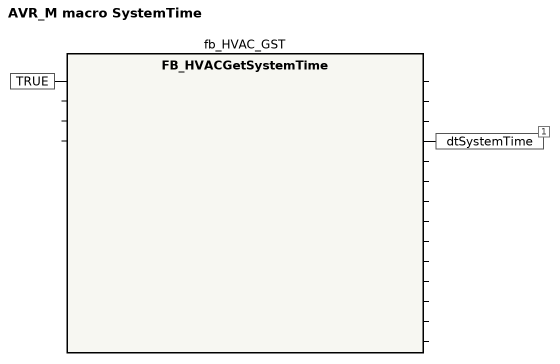
_CFC_ (* Continuous Function Chart, elements in execution order *)
#0 AND(SCHU_P2_2_UST_RE_PUSK, NOT SCHU_P2_2_YA1_DI6_ZKR)
#1 RT_T:R_TRIG(CLK: TRUE)
#2 OR(#1.Q, SCHU_P2_2_AVR_KOM_A)
#3 OR(SCHU_P2_2_AVR_KOM_M, NOT SCHU_P2_2_SA8_DI3_A, NOT SCHU_P2_2_SA1_DI5_A)
#4 TON_VKL:TON(IN: #3, PT: T#100ms)
#5 RS_avr_kom:RS(SET: #2, RESET1: #4.Q)
#6 TON_PUSK:TON(IN: #0, PT: t#6S)
#7 RT_Pusk:R_TRIG(CLK: #6.Q)
#8 OR(SCHU_P2_2_UST_RE_STOP, SCHU_P2_2_UST_RE_OSTANOV)
#9 RS_Pusk:RS(SET: #7.Q, RESET1: #8)
#10 SEL(#9.Q1, 0, 1)
#11 fb_HVACRC:FB_HVACRedundancyCtrl(EN: #5.Q1, eHVACDataSecurityType_Idle, FALSE, #10, NOT M1_OTKAZ, NOT M2_OTKAZ, -, -, -, -, -, -, SCHU_P2_2_MP2_2_1_DI3_RUN, SCHU_P2_2_MP2_2_2_DI7_RUN, -, -, -, -, -, -, -, dtSystemTime, -, SCHU_P2_2_M_SB_NAR, SCHU_P2_2_M_SB_NAR, SCHU_P2_2_SB, rHours, uiCount, overlap1Actuator, maxOnLevel, delayFBC)
#12 S SCHU_P2_2_AVR_A <= #11.ENO
#13 error <= #11.out 10
#14 NOT(#11.ENO)
#15 R SCHU_P2_2_AVR_A <= #14
#16 SCHU_P2_2_AVR_M <= #14
#17 AND(#11.ENO, #11.out 1)
#18 M1_PUSK <= #17
#19 AND(#11.ENO, #11.out 2)
#20 M2_PUSK <= #19
#21 MACRO SystemTime()
	#22 fb_HVAC_GST:FB_HVACGetSystemTime(TRUE, -, -, -)
	#23 dtSystemTime <= #22.out 4
END_MACRO
_END_CFC_
END_PROGRAM

(* POU TZBiS/TZB/Z_GVS1_Otk, CFC *)
PROGRAM Z_GVS1_Otk
VAR
	TON_YA2_OTKAZ: TON;
	SR_GVS1_Otkaz: SR;
	TON_YA2_Z_ZAM: TON;
END_VAR
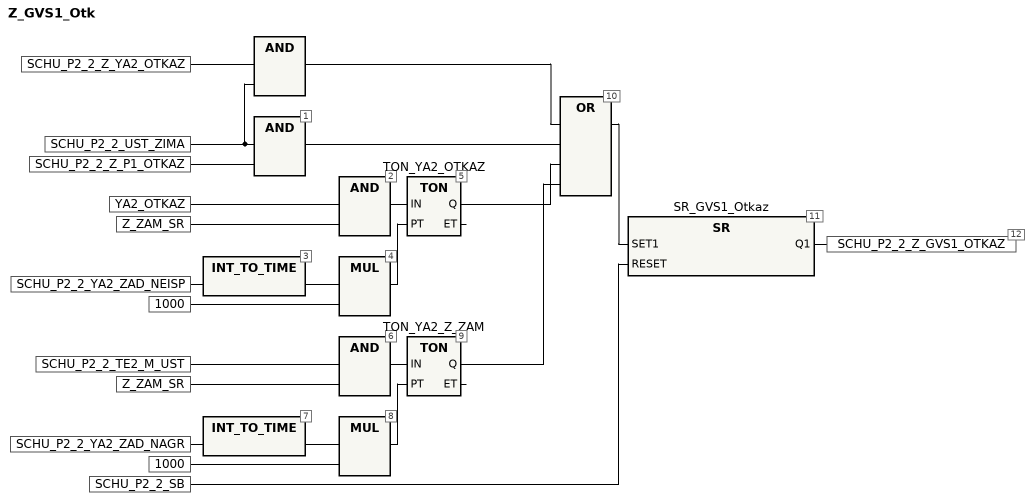
_CFC_ (* Continuous Function Chart, elements in execution order *)
#0 AND(SCHU_P2_2_Z_YA2_OTKAZ, SCHU_P2_2_UST_ZIMA)
#1 AND(SCHU_P2_2_UST_ZIMA, SCHU_P2_2_Z_P1_OTKAZ)
#2 AND(YA2_OTKAZ, Z_ZAM_SR)
#3 INT_TO_TIME(SCHU_P2_2_YA2_ZAD_NEISP)
#4 MUL(#3, 1000)
#5 TON_YA2_OTKAZ:TON(IN: #2, PT: #4)
#6 AND(SCHU_P2_2_TE2_M_UST, Z_ZAM_SR)
#7 INT_TO_TIME(SCHU_P2_2_YA2_ZAD_NAGR)
#8 MUL(#7, 1000)
#9 TON_YA2_Z_ZAM:TON(IN: #6, PT: #8)
#10 OR(#0, #1, #5.Q, #9.Q)
#11 SR_GVS1_Otkaz:SR(SET1: #10, RESET: SCHU_P2_2_SB)
#12 SCHU_P2_2_Z_GVS1_OTKAZ <= #11.Q1
_END_CFC_
(* the same logic as Structured Text *)
TON_YA2_OTKAZ(IN := YA2_OTKAZ AND Z_ZAM_SR, PT := INT_TO_TIME(SCHU_P2_2_YA2_ZAD_NEISP) * 1000);
TON_YA2_Z_ZAM(IN := SCHU_P2_2_TE2_M_UST AND Z_ZAM_SR, PT := INT_TO_TIME(SCHU_P2_2_YA2_ZAD_NAGR) * 1000);
SR_GVS1_Otkaz(SET1 := (SCHU_P2_2_Z_YA2_OTKAZ AND SCHU_P2_2_UST_ZIMA) OR (SCHU_P2_2_UST_ZIMA AND SCHU_P2_2_Z_P1_OTKAZ) OR TON_YA2_OTKAZ.Q OR TON_YA2_Z_ZAM.Q, RESET := SCHU_P2_2_SB);
SCHU_P2_2_Z_GVS1_OTKAZ := SR_GVS1_Otkaz.Q1;
END_PROGRAM

(* POU TZBiS/TZB/Z_M1_Avar, CFC *)
PROGRAM Z_M1_Avar
VAR
	SR_M1_Avar: SR;
END_VAR
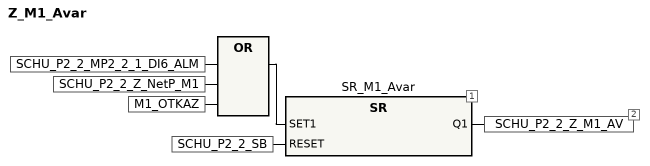
_CFC_ (* Continuous Function Chart, elements in execution order *)
#0 OR(SCHU_P2_2_MP2_2_1_DI6_ALM, SCHU_P2_2_Z_NetP_M1, M1_OTKAZ)
#1 SR_M1_Avar:SR(SET1: #0, RESET: SCHU_P2_2_SB)
#2 SCHU_P2_2_Z_M1_AV <= #1.Q1
_END_CFC_
(* the same logic as Structured Text *)
SR_M1_Avar(SET1 := SCHU_P2_2_MP2_2_1_DI6_ALM OR SCHU_P2_2_Z_NetP_M1 OR M1_OTKAZ, RESET := SCHU_P2_2_SB);
SCHU_P2_2_Z_M1_AV := SR_M1_Avar.Q1;
END_PROGRAM

(* POU TZBiS/TZB/Z_M1_NP, CFC *)
PROGRAM Z_M1_NP
VAR
	SR_M1_NPit: SR;
END_VAR
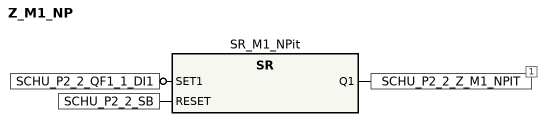
_CFC_ (* Continuous Function Chart, elements in execution order *)
#0 SR_M1_NPit:SR(SET1: NOT SCHU_P2_2_QF1_1_DI1, RESET: SCHU_P2_2_SB)
#1 SCHU_P2_2_Z_M1_NPIT <= #0.Q1
_END_CFC_
(* the same logic as Structured Text *)
SR_M1_NPit(SET1 := NOT SCHU_P2_2_QF1_1_DI1, RESET := SCHU_P2_2_SB);
SCHU_P2_2_Z_M1_NPIT := SR_M1_NPit.Q1;
END_PROGRAM

(* POU TZBiS/TZB/Z_M1_Pereg, CFC *)
PROGRAM Z_M1_Pereg
VAR
	SR_SCHU_P2_2_TSMP2_2_1_DI7: SR;
	TOF_TSMP1: TOF;
	TON1: TON;
END_VAR
VAR (* helpers for the ST form of the networks *)
	_t23 : BOOL;
END_VAR
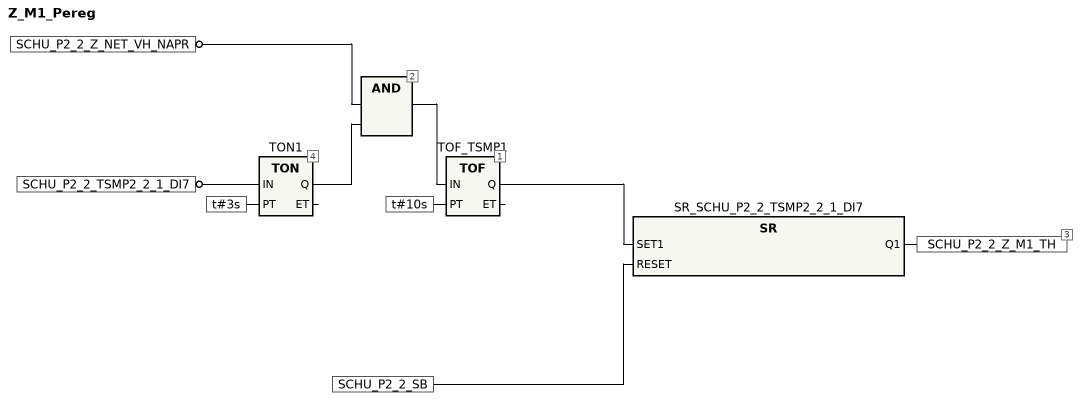
_CFC_ (* Continuous Function Chart, elements in execution order *)
#0 SR_SCHU_P2_2_TSMP2_2_1_DI7:SR(SET1: #1.Q, RESET: SCHU_P2_2_SB)
#1 TOF_TSMP1:TOF(IN: #2, PT: t#10s)
#2 AND(NOT SCHU_P2_2_Z_NET_VH_NAPR, #4.Q)
#3 SCHU_P2_2_Z_M1_TH <= #0.Q1
#4 TON1:TON(IN: NOT SCHU_P2_2_TSMP2_2_1_DI7, PT: t#3s)
_END_CFC_
(* the same logic as Structured Text *)
SR_SCHU_P2_2_TSMP2_2_1_DI7(SET1 := TOF_TSMP1.Q, RESET := SCHU_P2_2_SB);
TOF_TSMP1(IN := _t23, PT := t#10s);
_t23 := NOT SCHU_P2_2_Z_NET_VH_NAPR AND TON1.Q;
SCHU_P2_2_Z_M1_TH := SR_SCHU_P2_2_TSMP2_2_1_DI7.Q1;
TON1(IN := NOT SCHU_P2_2_TSMP2_2_1_DI7, PT := t#3s);
END_PROGRAM

(* POU TZBiS/TZB/Z_M2_Avar, CFC *)
PROGRAM Z_M2_Avar
VAR
	SR_M2_Avar: SR;
END_VAR
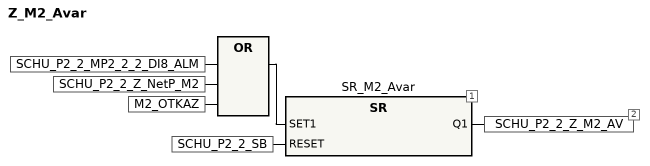
_CFC_ (* Continuous Function Chart, elements in execution order *)
#0 OR(SCHU_P2_2_MP2_2_2_DI8_ALM, SCHU_P2_2_Z_NetP_M2, M2_OTKAZ)
#1 SR_M2_Avar:SR(SET1: #0, RESET: SCHU_P2_2_SB)
#2 SCHU_P2_2_Z_M2_AV <= #1.Q1
_END_CFC_
(* the same logic as Structured Text *)
SR_M2_Avar(SET1 := SCHU_P2_2_MP2_2_2_DI8_ALM OR SCHU_P2_2_Z_NetP_M2 OR M2_OTKAZ, RESET := SCHU_P2_2_SB);
SCHU_P2_2_Z_M2_AV := SR_M2_Avar.Q1;
END_PROGRAM

(* POU TZBiS/TZB/Z_M2_NP, CFC *)
PROGRAM Z_M2_NP
VAR
	SR_M2_NPit: SR;
END_VAR
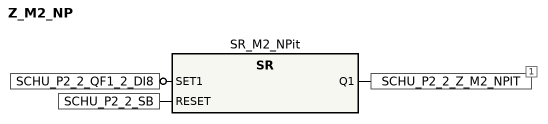
_CFC_ (* Continuous Function Chart, elements in execution order *)
#0 SR_M2_NPit:SR(SET1: NOT SCHU_P2_2_QF1_2_DI8, RESET: SCHU_P2_2_SB)
#1 SCHU_P2_2_Z_M2_NPIT <= #0.Q1
_END_CFC_
(* the same logic as Structured Text *)
SR_M2_NPit(SET1 := NOT SCHU_P2_2_QF1_2_DI8, RESET := SCHU_P2_2_SB);
SCHU_P2_2_Z_M2_NPIT := SR_M2_NPit.Q1;
END_PROGRAM

(* POU TZBiS/TZB/Z_M2_Pereg, CFC *)
PROGRAM Z_M2_Pereg
VAR
	SR_SCHU_P2_2_TSMP2_2_2_DI1: SR;

	TOF_TSMP2: TOF;
	TON1: TON;
END_VAR
VAR (* helpers for the ST form of the networks *)
	_t28 : BOOL;
END_VAR
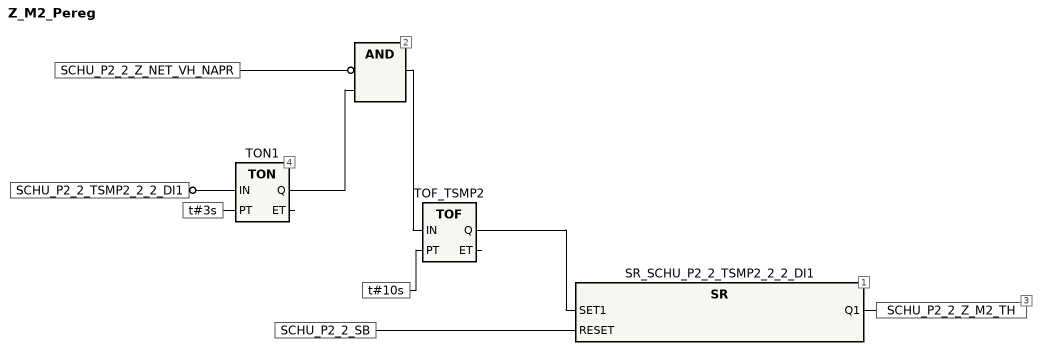
_CFC_ (* Continuous Function Chart, elements in execution order *)
#0 TOF_TSMP2:TOF(IN: #2, PT: t#10s)
#1 SR_SCHU_P2_2_TSMP2_2_2_DI1:SR(SET1: #0.Q, RESET: SCHU_P2_2_SB)
#2 AND(NOT SCHU_P2_2_Z_NET_VH_NAPR, #4.Q)
#3 SCHU_P2_2_Z_M2_TH <= #1.Q1
#4 TON1:TON(IN: NOT SCHU_P2_2_TSMP2_2_2_DI1, PT: t#3s)
_END_CFC_
(* the same logic as Structured Text *)
TOF_TSMP2(IN := _t28, PT := t#10s);
SR_SCHU_P2_2_TSMP2_2_2_DI1(SET1 := TOF_TSMP2.Q, RESET := SCHU_P2_2_SB);
_t28 := NOT SCHU_P2_2_Z_NET_VH_NAPR AND TON1.Q;
SCHU_P2_2_Z_M2_TH := SR_SCHU_P2_2_TSMP2_2_2_DI1.Q1;
TON1(IN := NOT SCHU_P2_2_TSMP2_2_2_DI1, PT := t#3s);
END_PROGRAM

(* POU TZBiS/TZB/Z_NET_VKH_NAPR, CFC *)
PROGRAM Z_NET_VKH_NAPR
VAR
	RS_Net_vhk_napr: SR;
END_VAR
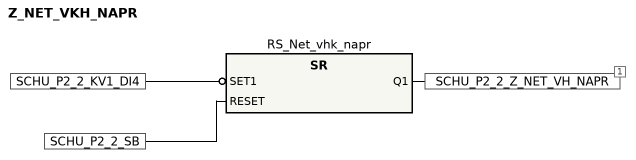
_CFC_ (* Continuous Function Chart, elements in execution order *)
#0 RS_Net_vhk_napr:SR(SET1: NOT SCHU_P2_2_KV1_DI4, RESET: SCHU_P2_2_SB)
#1 SCHU_P2_2_Z_NET_VH_NAPR <= #0.Q1
_END_CFC_
(* the same logic as Structured Text *)
RS_Net_vhk_napr(SET1 := NOT SCHU_P2_2_KV1_DI4, RESET := SCHU_P2_2_SB);
SCHU_P2_2_Z_NET_VH_NAPR := RS_Net_vhk_napr.Q1;
END_PROGRAM

(* POU TZBiS/TZB/Z_NP, CFC *)
PROGRAM Z_NP
VAR
	TON_PDS2: TON;
	TON_ReRab: TON;
	TON_MVKL: TON;
	TON_AVT: TON;
	TP_SR: TP;
	SR_NP_M1: SR;
	SR_NP_M2: SR;
	TON_MVKL_M1: TON;
	TON_AVT_M1: TON;
	TON_AVT_M2: TON;
	TON_MVKL_M2: TON;
END_VAR
VAR (* helpers for the ST form of the networks *)
	_t70 : BOOL;
END_VAR
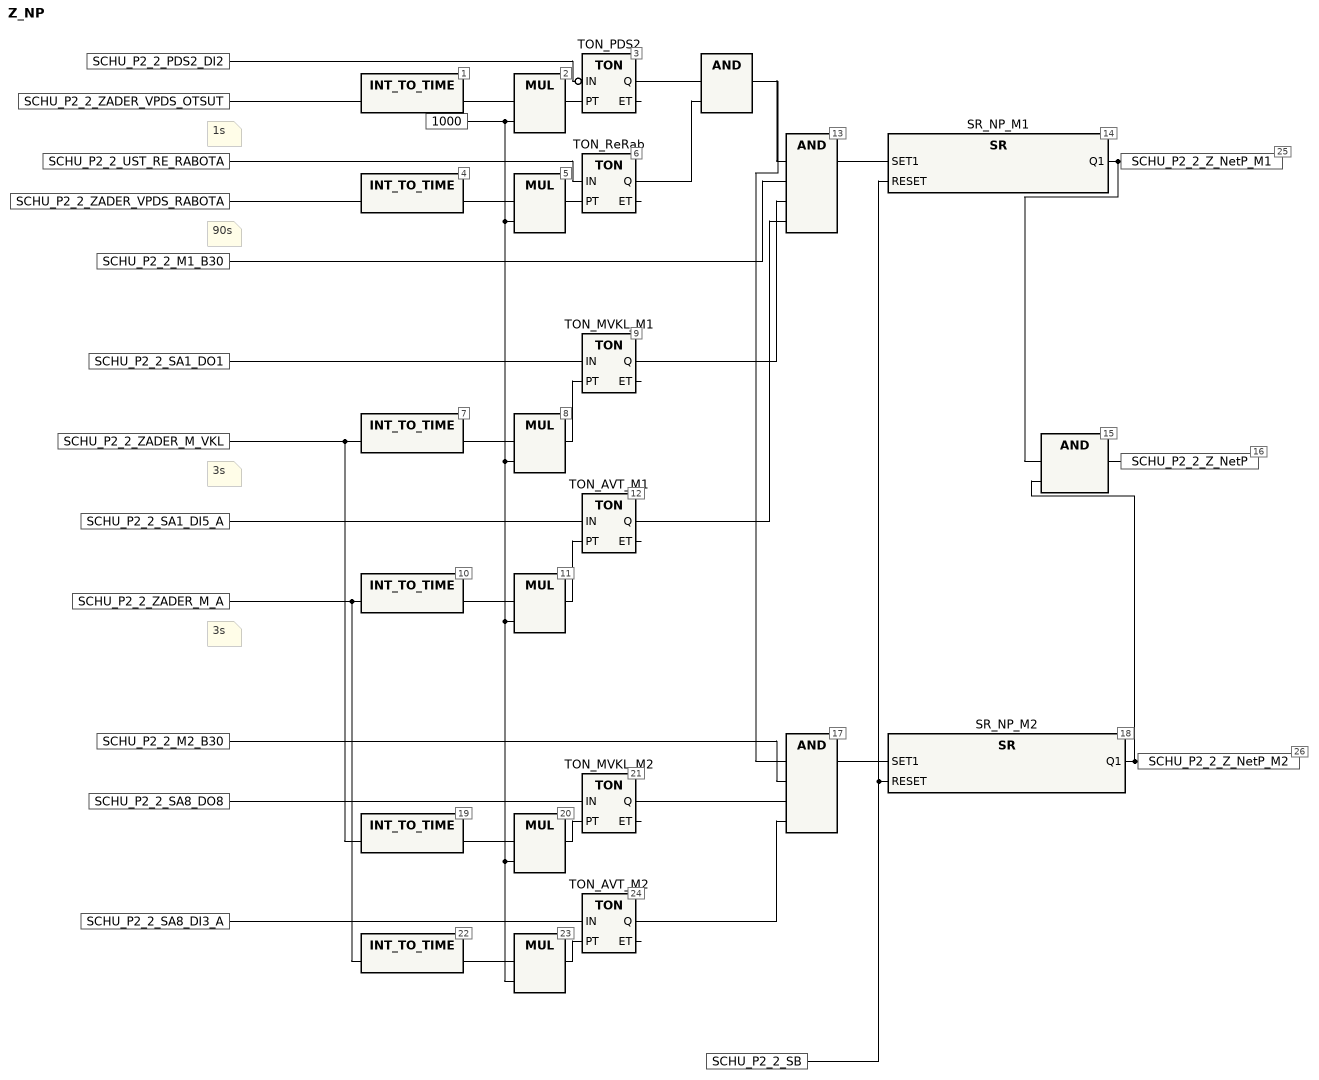
